Staubli VAL3: ManualJoint.pgx

program ManualJoint()
begin
  jHere = herej()
  OPCj1cmd = jHere.j1
  OPCj2cmd = jHere.j2
  OPCj3cmd = jHere.j3
  OPCj4cmd = jHere.j4
  OPCj5cmd = jHere.j5
  OPCj6cmd = jHere.j6

  while true
    jJointRx.j1=OPCj1cmd
    jJointRx.j2=OPCj2cmd
    jJointRx.j3=OPCj3cmd
    jJointRx.j4=OPCj4cmd
    jJointRx.j5=OPCj5cmd
    jJointRx.j6=OPCj6cmd
    movej(jJointRx,flange,mAppro)
    waitEndMove()
  endWhile
end
